VAR_GLOBAL
END_VAR

(* stored: Version 1.1.0.1, ProductVersion 3.1.4022.12
   GVL etsitaan: Id {1e3d9884-7ae7-4456-912a-3e02fa1fff28} *)
